Staubli VAL3: reset.pgx

public program reset()
begin
  // This program resets the encoder librarie. This reset consist of
  //  - resetting the VAL3 counter
  //  - Resetting the digital output cRstErr
  // This actions are performed in the program "encoder" of the library
  // Created 29-05-08                                  C.CURRIVAND
  //----------------------------------------------------------------
  bReset=true
end
